{attribute 'analysis' := '-27'}
VAR_GLOBAL

	fbTestsuites:			FB_Testsuites;				// Testsuites
END_VAR

(* stored: Version 1.1.0.1
   GVL GVL: Id {ae26674a-b3aa-0ba1-1260-3c9013903e0e} *)
